// TIA Portal V17 export
// export: Created 2025-03-05T08:02:27.9727813Z, ExportSetting WithDefaults, DisplayName Totally Integrated Automation Portal, DisplayVersion V17 Update 8, DisplayName TIA Portal Openness, DisplayVersion V17 Update 8, DisplayName TIA Portal Version Control Interface, DisplayVersion V17, DisplayName SINAMICS Startdrive Advanced, DisplayVersion V17 SP2, DisplayName SINAMICS Startdrive G110M, G120, G120C, G120D, G120P, G115D, DisplayVersion V17 SP2, DisplayName SINAMICS Startdrive G130, G150, S120, S150, SINAMICS MV, S210, DisplayVersion V17 SP2, DisplayName STEP 7 Professional, DisplayVersion V17 Update 8, DisplayName SINUMERIK ONE STEP 7 Toolbox, DisplayVersion V17 Update 12, DisplayName SINUMERIK 840D sl STEP 7 Toolbox, DisplayVersion V17 Update 12, DisplayName STEP 7 Safety, DisplayVersion V17 Update 6, DisplayName WinCC Advanced, DisplayVersion V17 Update 8
TYPE "LASER POINTER"
// stored: IsFailsafeCompliant false
   STRUCT
      "LASER POINTER INPUT ON" : Bool;
      "LASER POINTER START GENERAL CONDITIONS" : Bool;
      "LASER POINTER START INITIAL CONDITIONS" : Bool;
      "LASER POINTER MANUAL START REQUEST" : Bool;
      "LASER POINTER AUTO START REQUEST" : Bool;
      "LASER POINTER START REQUEST" : Bool;
      "LASER POINTER START COMMAND" : Bool;
      "LASER POINTER LASER SYSTEM ON" : Bool;
      "LASER POINTER FEEDBACK ON" : Bool;
      "LASER POINTER STOP GENERAL CONDITIONS" : Bool;
      "LASER POINTER STOP INITIAL CONDITIONS" : Bool;
      "LASER POINTER MANUAL STOP REQUEST" : Bool;
      "LASER POINTER AUTO STOP REQUEST" : Bool;
      "LASER POINTER STOP REQUEST" : Bool;
      "LASER POINTER STOP COMMAND" : Bool;
      "LASER POINTER STOPPED" : Bool;
      "LASER POINTER FEEDBACK OFF" : Bool;
      "LASER POINTER WARNING GONE" : Bool;
      "LASER POINTER START GENERAL CONDITION HELP" : Bool;
      "LASER POINTER START INITIAL CONDITION HELP" : Bool;
      "LASER POINTER STOP GENERAL CONDITION HELP" : Bool;
      "LASER POINTER STOP INITIAL CONDITION HELP" : Bool;
      "LASER POINTER NOT READY ALARM" : Bool;
      "LASER POINTER FAULT" : Bool;
   END_STRUCT;
END_TYPE
